PROGRAM MAIN
VAR
END_VAR

END_PROGRAM

(* stored: Version 1.1.0.1
   POU MAIN: Id {b086714b-4cee-446e-861a-7a5196c9958e} *)
